PROGRAM MAIN
VAR
	fbServerClientConnection : FB_ServerClientConnection;
	fbSocketSend : FB_SocketSend;
	fbSocketReceive : FB_SocketReceive;
	hServer : T_HSERVER; 
	
	bInit : BOOL := TRUE;
	
	ePhase : E_ServerPhases := INIT_PHASE;
	receiveBuffer : T_MAXSTRING;
END_VAR

F_CreateServerHnd(
	sSrvNetID := '127.0.0.1.1.1',
	sLocalHost := '',
	nLocalPort := 200,
	nMode :=  LISTEN_MODE_CLOSEALL,
	bEnable := bInit,
	hServer := hServer);

fbServerClientConnection(
	hServer := hServer,
	bEnable := NOT bInit,
	nRemotePort := 80,
	tReconnect := T#30MS);

fbSocketReceive(
	bExecute := (ePhase = RECEIVE_PHASE),
	tTimeout := T#30S,
	pDest := ADR(receiveBuffer),
	cbLen := SIZEOF(receiveBuffer),
	hSocket := fbServerClientConnection.hSocket);
	
	
CASE ePhase OF

	INIT_PHASE:
		bInit := FALSE;
		ePhase := START_PHASE;
		
	START_PHASE:
		IF fbServerClientConnection.eState = E_SocketConnectionState.eSOCKET_CONNECTED THEN
			ePhase := RECEIVE_PHASE;
		END_IF
		
	RECEIVE_PHASE:
		
		
END_CASE

END_PROGRAM

(* stored: Version 1.1.0.1, ProductVersion 3.1.4024.4
   POU MAIN: Id {fe4c4bd0-bb2f-4c2f-8bc6-e4fda118c397}, SpecialFunc None *)
